Staubli VAL3: MIDPOS.pgx

public program midPos(string x_sItem, num x_nLength, num x_nPos, string& x_sResult[])
  local string l_sLeft
begin
  //-----------------------------------------------------------------------
  //Header begin
  //Description of program
  //  This program allows to keep x_nLength characters of a string from
  //  a position x_nPos.
  //  The characters before and after x_nPos and x_nPos+x_nLength will be
  //  truncated.
  //
  //Input parameters
  //  string x_sItem :
  //    role : string that you wan to cut
  //  num x_nLength :
  //    role : Length of the characters that you want to keep
  //  num x_nPos :
  //    role : Position to start keeping characters
  //
  //Output parameters
  //  string x_sResult :
  //    role : string truncated
  //
  //Example
  //  call midPos("Staubli Robotics",4,2,sResult)
  //  put(sResult) //Displays "aubl"
  //
  //History
  //  Creation : 28-04-08 - f.Rob
  //Header end
  //-----------------------------------------------------------------------
  // LEFT SIDE
  call leftPos(x_sItem,x_nLength+x_nPos,l_sLeft)
  // update
  x_sResult=l_sLeft
  // RIGHT SIDE
  call rightPos(l_sLeft,x_nLength,x_sResult)
  // OK ....
end
